INTERFACE I_ErrorHandling

PROPERTY P_Error : bool
GET
END_GET
END_PROPERTY

PROPERTY P_ErrorID : udint
GET
END_GET
END_PROPERTY

METHOD ToString : String(255)
VAR_INPUT
END_VAR
END_METHOD

END_INTERFACE

(* stored: Version 1.1.0.1, ProductVersion 3.1.4022.12
   Itf I_ErrorHandling: Id {da216883-1660-4181-8363-d7bbed513f94}
   Property P_Error: Id {2bb939aa-a95e-454f-a6d7-d1d817398b7a}
   Get Get: Id {e8aa9bbc-3388-4f63-b995-747841c7ae25}
   Property P_ErrorID: Id {a105f56c-fd7d-4285-a6bc-da3fa6a15c52}
   Get Get: Id {697f4561-6929-4c35-a4e4-26ff7b85b532}
   Method ToString: Id {7c2321d9-78d6-4ab4-b395-3241892617ac} *)
